// TIA Portal V14 SP1 export
// export: Created 2019-05-02T00:21:54.0023896Z, ExportSetting WithReadOnly, DisplayName Totally Integrated Automation Portal, DisplayVersion V14 SP1 Update 7, DisplayName TIA Portal Openness, DisplayVersion V14 SP1 Update 6, DisplayName STEP 7 Basic, DisplayVersion V14 SP1 Update 7, DisplayName WinCC Basic, DisplayVersion V14 SP1 Update 7
ORGANIZATION_BLOCK "Main"   // OB1, LAD, ProgramCycle
TITLE = "Main Program Sweep (Cycle)"
{ S7_Optimized_Access := 'TRUE' }
// stored: CodeModifiedDate 2019-05-02T00:19:22.0356737Z, CompileDate 2019-05-02T00:21:49.3422341Z, CreationDate 2019-05-02T00:12:13.7630248Z, InterfaceModifiedDate 2008-07-21T16:55:08.419547Z, IsConsistent true, ModifiedDate 2019-05-02T00:19:22.0356737Z, ParameterModified 2008-07-21T16:55:08.419547Z, StructureModified 2008-07-21T16:55:08.419547Z
   VAR_INPUT
      Initial_Call : Bool;   // Initial call of this OB
      Remanence : Bool;   // =True, if remanent data are available
   END_VAR
BEGIN

REGION Network 1
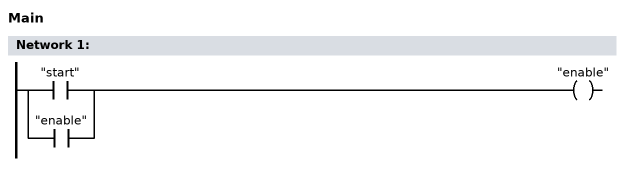
   RUNG wire#powerrail
      Contact( "start" )
      wire#w1
      Coil( "enable" )
   END_RUNG
   RUNG wire#powerrail
      Contact( "enable" )
   END_RUNG wire#w1
   // the same network as SCL:
   "enable" := "start" OR "enable";
END_REGION
END_ORGANIZATION_BLOCK
